// TIA Portal V15.1 export
// export: Created 2019-08-08T13:58:53.505237Z, ExportSetting None, DisplayName Totally Integrated Automation Portal, DisplayVersion V15.1, DisplayName TIA Portal Openness, DisplayVersion V15.1, DisplayName STEP 7 Professional, DisplayVersion V15.1, DisplayName STEP 7 Safety, DisplayVersion V15.1, DisplayName WinCC Advanced, DisplayVersion V15.1
TYPE "typeModulSkillInterface_IN"
   STRUCT
      Enable : Bool;
      Init : Bool;
      Reset : Bool;
      Manual : Bool;
      Automatic : Bool;
      SingleStep : Bool;
      Start : Bool;
      "Step" : Bool;
      Stop : Bool;
   END_STRUCT;
END_TYPE
